FUNCTION_BLOCK FB_ManipAxis
VAR_INPUT
END_VAR
VAR_OUTPUT
	q_asResult: ARRAY [1..20] OF STRING;
	q_xError	:	BOOL;
END_VAR
VAR_IN_OUT
	iq_ManipAxis	:	ST_ManipAxis;
END_VAR
VAR
	

	mcPower	:	MC_Power;
	mcReset	:	MC_Reset;
	mcMoveAbsolute : ARRAY[1..2] OF MC_MoveAbsolute;
	mcHalt	:	MC_Halt;
	
	//Error Stuff
	indexResult: INT := 1;
	fbFormatString	:	FB_FormatString;
	
	xInitComplete	:	BOOL := FALSE;
	
	imcBlockIndex: INT;
	imcBlockIndexPrev : INT;
	
	rtEnable : R_TRIG;
	ftEnable : F_TRIG;
	rtStop	:	R_TRIG;
	rtStart	:	R_TRIG;
	rReqAbsPosOld: REAL := 0;
	rReqAbsPosPrevious: REAL;
	iI: INT;
END_VAR

(* Manipulator Axis Function Block
Alex Wallace, 2016-8-8 


*)


rtEnable(CLK:=iq_ManipAxis.xEnable);
ftEnable(CLK:=iq_ManipAxis.xEnable);

//Update status
iq_ManipAxis.stAxis();

IF rtEnable.Q OR ftEnable.Q THEN
	xInitComplete := FALSE;
	iq_ManipAxis.eState := Init;
ELSIF xInitComplete THEN
	iq_ManipAxis.eState := MoveEnabled;
END_IF

//Restart a move
rtStart(CLK:=iq_ManipAxis.xStart);

//For EPICS, because the modbus map was made for 32 bit..
iq_ManipAxis.rActPos := LREAL_TO_REAL(iq_ManipAxis.stAxis.NcToPlc.ActPos);


CASE iq_ManipAxis.eState OF
	0: iq_ManipAxis.eState := Init;
	Init:
	(* Start by initializing the motor axis *)
	mcPower.Enable := iq_ManipAxis.xEnable;
	
	IF mcPower.Status THEN //success
		xInitComplete := TRUE;
		q_asResult[indexResult] := 'Motor init success';
		indexResult := indexResult + 1;
		iq_ManipAxis.eState := MoveEnabled;
	ELSIF mcPower.Error THEN
		mcPower.Enable := FALSE;
		fbFormatString(sFormat:='Init mcPower Error: %s', arg1:=F_UDINT(mcPower.ErrorID));
		ActError();
	END_IF
		
	MoveEnabled:
		IF (iq_ManipAxis.rReqAbsPos <> rReqAbsPosPrevious OR rtStart.Q)  AND iq_ManipAxis.xEnable THEN
			mcMoveAbsolute[imcBlockIndex].Execute := FALSE;
			imcBlockIndex := imcBlockIndex + 1;
			IF imcBlockIndex >2 THEN imcBlockIndex := 1; END_IF
			mcMoveAbsolute[imcBlockIndex].Position := LIMIT(0, REAL_TO_LREAL(iq_ManipAxis.rReqAbsPos), 100);
			mcMoveAbsolute[imcBlockIndex].Execute := TRUE;
			rReqAbsPosPrevious := iq_ManipAxis.rReqAbsPos;
		ELSIF mcMoveAbsolute[imcBlockIndex].Done OR mcMoveAbsolute[imcBlockIndex].CommandAborted OR mcMoveAbsolute[imcBlockIndex].Busy OR mcMoveAbsolute[imcBlockIndex].Error THEN
			mcMoveAbsolute[imcBlockIndex].Execute := FALSE;
			iq_ManipAxis.xStart := FALSE;
		END_IF
		//Halt
		mcHalt.Execute S= iq_ManipAxis.xStop;
		mcHalt.Execute R= mcHalt.Busy;
		iq_ManipAxis.xStop R= mcHalt.Busy;

	Error:
		mcReset.Execute := rtEnable.Q;
		IF mcReset.Done THEN
			q_xError := FALSE;
			mcReset.Execute := FALSE;
			iq_ManipAxis.eState:=Init;
		END_IF
	
END_CASE


(* Run the mc blocks *)
ActPower();
mcReset(Axis:=iq_ManipAxis.stAxis);
mcHalt(Axis:=iq_ManipAxis.stAxis);
FOR iI := 1 TO 2 DO
mcMoveAbsolute[iI](Axis := iq_ManipAxis.stAxis, Velocity:=iq_ManipAxis.lrVelocity, BufferMode:=MC_Aborting);
END_FOR

ACTION ActPower:
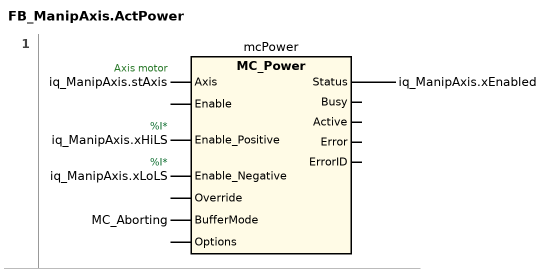
// NETWORK 1
//   iq_ManipAxis.stAxis: Axis motor
//   iq_ManipAxis.xHiLS: AT %I*
//   iq_ManipAxis.xLoLS: AT %I*
mcPower(
    Axis := iq_ManipAxis.stAxis,
    Enable_Positive := iq_ManipAxis.xHiLS,
    Enable_Negative := iq_ManipAxis.xLoLS,
    BufferMode := MC_Aborting); // MC_Power
iq_ManipAxis.xEnabled := mcPower.Status;
END_ACTION

ACTION ActError:
(* Error action
*)

//Reset the debugging index
IF indexResult > 20 THEN indexResult := 1; END_IF

iq_ManipAxis.eState := Error;
q_xError	:=	TRUE;
q_asResult[indexResult] := fbFormatString.sOut;
indexResult := indexResult +1;
END_ACTION

END_FUNCTION_BLOCK

(* stored: Version 1.1.0.1, ProductVersion 3.1.4020.12
   POU FB_ManipAxis: Id {2c576ec6-7433-4ec0-8547-ab9b5dd393c9}, SpecialFunc None
   Action ActPower: Id {31b74a81-1b68-4db8-b9a3-64793fff0f5a}
   Action ActError: Id {efb14a67-3fcd-4d5f-a82f-60b8d6779b53} *)
